{attribute 'Tc2GvlVarNames'}
VAR_GLOBAL
	
(*Pnc_Chariot*)
	Fonction_Abaissement_Relevage_Pince		:BOOL;
	
(*Pnc_Operateur*)
	Option_Detection_Pince					:BOOL:=FALSE;	
	Fonction_arret_Centrale_automatique		:BOOL:=FALSE;

(*Pnc_Vernet*)
	Chariot_a_Gauche						:BOOL:=TRUE;
	Type_Machine_VP							:BOOL:=FALSE;
                                    	
(*Pnc_Free_Bool*)                   	
	Maintenance								:BOOL:=FALSE;
                                    	

END_VAR

(* stored: Version 1.1.0.1, ProductVersion 3.1.4024.15
   GVL Global_Configuration_Machine_PNC: Id {30407aef-336f-40bf-831c-f6beea47fb9b} *)
